(* IEC 61131-3 sources: altus-mobile/clpaltus/codigo/clp_mestre, 3 files *)

(* ---- GVL_MODBUS.st ---- *)
(*
  ARQUIVO: GVL_MODBUS.st — CLP MESTRE (gateway)
  ONDE USAR: MasterTool > Application > UserGVLs > GVL_MODBUS
  O QUE FAZ: registradores Modbus do mestre.

  DIREÇÃO DOS REGISTRADORES:
    MB_CMD_*  → mestre ESCREVE no escravo  (FC16 - Write Multiple Registers)
                  contém os comandos recebidos do app via MQTT
    MB_FB_*   → mestre LÊ do escravo       (FC03 - Read Holding Registers)
                  contém o estado real das saídas executadas pelo escravo

  ENDEREÇOS NO ESCRAVO:
    MB_CMD_KIT1 → Holding Register 40001 (endereço 0)
    MB_CMD_KIT2 → Holding Register 40002 (endereço 1)
    MB_FB_KIT1  → Holding Register 40003 (endereço 2)
    MB_FB_KIT2  → Holding Register 40004 (endereço 3)
*)

VAR_GLOBAL

    (* --- COMANDOS: mestre envia ao escravo (app → mestre → escravo) --- *)
    (* Cada bit representa uma saída. Bit 0 = Kit1/pushbutton/1, etc. *)
    MB_CMD_KIT1 : WORD;   (* bits 0-7: CMD_Q00 a CMD_Q07 *)
    MB_CMD_KIT2 : WORD;   (* bits 0-7: CMD_Q08 a CMD_Q15 *)

    (* --- RETORNO: mestre lê do escravo (escravo → mestre → app) --- *)
    (* Preenchido pelo escravo com o estado real das saídas físicas *)
    MB_FB_KIT1  : WORD;   (* bits 0-7: estado real Q00-Q07 no escravo *)
    MB_FB_KIT2  : WORD;   (* bits 0-7: estado real Q08-Q15 no escravo *)

    (* Comandos individuais (BOOL) — preenchidos pelo MQTT_RECEBER *)
    CMD_Q00 : BOOL;   CMD_Q01 : BOOL;   CMD_Q02 : BOOL;   CMD_Q03 : BOOL;
    CMD_Q04 : BOOL;   CMD_Q05 : BOOL;   CMD_Q06 : BOOL;   CMD_Q07 : BOOL;
    CMD_Q08 : BOOL;   CMD_Q09 : BOOL;   CMD_Q10 : BOOL;   CMD_Q11 : BOOL;
    CMD_Q12 : BOOL;   CMD_Q13 : BOOL;   CMD_Q14 : BOOL;   CMD_Q15 : BOOL;

END_VAR

(* ---- GVL_MQTT.st ---- *)
(*
  ARQUIVO: GVL_MQTT.st — CLP MESTRE (gateway)
  ONDE USAR: MasterTool > Application > UserGVLs > GVL_MQTT
  O QUE FAZ: variáveis MQTT do CLP mestre.
             O mestre só recebe comandos do app e publica o retorno do escravo.
             Quem executa as saídas físicas é o CLP escravo.
*)

VAR_GLOBAL

    (* Arrays internos da biblioteca LibMQTT — não mexa *)
    Pubs : ARRAY[1..gc_uiMaxPubs] OF MQTT_PUBLISH;
    Subs : ARRAY[1..gc_uiMaxSubs] OF MQTT_SUBSCRIBE;

    (* 16 tópicos — os mesmos para receber (subscribe) e publicar retorno (publish) *)
    MQTT_TOPICS : ARRAY[1..16] OF STRING := [
        'altus/kit1/pushbutton/1',   (* pos 1  → CMD_Q00 / kit1Led1 *)
        'altus/kit1/pushbutton/2',   (* pos 2  → CMD_Q01 / kit1Led2 *)
        'altus/kit1/pushbutton/3',   (* pos 3  → CMD_Q02 / kit1Led3 *)
        'altus/kit1/pushbutton/4',   (* pos 4  → CMD_Q03 / kit1Led4 *)
        'altus/kit1/switch/1',       (* pos 5  → CMD_Q04 / kit1Led5 *)
        'altus/kit1/switch/2',       (* pos 6  → CMD_Q05 / kit1Led6 *)
        'altus/kit1/switch/3',       (* pos 7  → CMD_Q06 / kit1Led7 *)
        'altus/kit1/switch/4',       (* pos 8  → CMD_Q07 / kit1Led8 *)
        'altus/kit2/pushbutton/1',   (* pos 9  → CMD_Q08 / kit2Led1 *)
        'altus/kit2/pushbutton/2',   (* pos 10 → CMD_Q09 / kit2Led2 *)
        'altus/kit2/pushbutton/3',   (* pos 11 → CMD_Q10 / kit2Led3 *)
        'altus/kit2/pushbutton/4',   (* pos 12 → CMD_Q11 / kit2Led4 *)
        'altus/kit2/switch/1',       (* pos 13 → CMD_Q12 / kit2Led5 *)
        'altus/kit2/switch/2',       (* pos 14 → CMD_Q13 / kit2Led6 *)
        'altus/kit2/switch/3',       (* pos 15 → CMD_Q14 / kit2Led7 *)
        'altus/kit2/switch/4'        (* pos 16 → CMD_Q15 / kit2Led8 *)
    ];

    (* O que chegou do app — payloads recebidos de cada tópico *)
    SUBS_PAYLOADS : ARRAY[1..gc_uiMaxSubs] OF STRING;

    (* O que vai publicar de volta — preenchido pelo MODBUS_GATEWAY com o retorno do escravo *)
    PUBS_PAYLOADS     : ARRAY[1..gc_uiMaxPubs] OF STRING;
    PUBS_PAYLOADS_OLD : ARRAY[1..gc_uiMaxPubs] OF STRING;

    (* Status internos *)
    MQTT_FB_Pub_Status        : ARRAY[1..gc_uiMaxPubs] OF BOOL;
    MQTT_FB_Received_Messages : ARRAY[1..gc_uiMaxSubs] OF MQTT_RECEIVED;

END_VAR

(* ---- MQTT.st ---- *)
(*
  ARQUIVO: MQTT.st — CLP MESTRE (gateway)
  ONDE USAR: MasterTool > pasta MQTT > MQTT (PRG)
  O QUE FAZ: mantém a conexão MQTT, assina os 16 tópicos do app
             e publica de volta o retorno do CLP escravo (para atualizar LEDs).

  TROQUE O IP: coloque o IP do PC onde o Mosquitto está rodando.
  Para descobrir: abra o CMD e digite "ipconfig" → "Endereço IPv4"
*)

(* ================================================================
   SEÇÃO VAR — cole na parte de CIMA do editor (área de variáveis)
   ================================================================ *)
(*
VAR
    MQTT_FB            : MQTT_CLIENT;
    MQTT_FB_Enable     : BOOL := TRUE;
    MQTT_FB_Error      : BOOL;
    MQTT_FB_State      : MQTT_STATES;
    MQTT_FB_Error_Code : MQTT_ERR_CODE;
    i                  : INT;
END_VAR
*)

(* ================================================================
   CÓDIGO — cole na parte de BAIXO do editor
   ================================================================ *)

(* ------ TROQUE O IP AQUI ------ *)
MQTT_FB_CONNECTION_CONFIG.sHostname     := '192.168.X.X';
MQTT_FB_CONNECTION_CONFIG.uiPort        := 1883;
MQTT_FB_CONNECTION_CONFIG.sClientId     := 'clp_mestre_gateway';
MQTT_FB_CONNECTION_CONFIG.bCleanSession := TRUE;

MQTT_FB.PUBLISH   := Pubs;
MQTT_FB.SUBSCRIBE := Subs;
MQTT_FB_Enable    := MQTT_FB.Enable;

MQTT_FB_Error             := MQTT_FB.ERROR;
MQTT_FB_State             := MQTT_FB.STATE;
MQTT_FB_Error_Code        := MQTT_FB.ERROR_CODE;
MQTT_FB_Pub_Status        := MQTT_FB.PUBLISH_STATUS;
MQTT_FB_Received_Messages := MQTT_FB.RECEIVED_MESSAGES;

(* Publicação: retorno do escravo → atualiza LEDs do app *)
FOR i := 1 TO 16 DO
    Pubs[i].sPublishTopic        := MQTT_TOPICS[i];
    Pubs[i].pbPublishPayload     := ADR(PUBS_PAYLOADS[i]);
    Pubs[i].uiPublishPayloadSize := TO_UINT(LEN(PUBS_PAYLOADS[i]));
    Pubs[i].uiPublishMessageQos  := MQTT_QOS_0;
    Pubs[i].bPublishRetain       := TRUE;

    IF (PUBS_PAYLOADS[i] <> PUBS_PAYLOADS_OLD[i]) THEN
        PUBS_PAYLOADS_OLD[i]     := PUBS_PAYLOADS[i];
        Pubs[i].bEnablePublish   := TRUE;
    END_IF

    IF (MQTT_FB_Pub_Status[i]) THEN
        Pubs[i].bEnablePublish   := FALSE;
    END_IF
END_FOR

(* Assinatura: recebe comandos do app *)
FOR i := 1 TO 16 DO
    Subs[i].eSubscribeTopic  := MQTT_TOPICS[i];
    Subs[i].pbPayloadBuffer  := ADR(SUBS_PAYLOADS[i]);
    Subs[i].uiMaxPayloadSize := SIZEOF(SUBS_PAYLOADS[i]);
    Subs[i].eSubscribeQos    := MQTT_QOS_0;
END_FOR

IF MQTT_FB_Error THEN
    MQTT_FB_Enable := PULSE_55;
ELSE
    MQTT_FB_Enable := TRUE;
END_IF

MQTT_FB();
